FUNCTION Convert_LWORD_TO_TOD : Hresult
VAR_INPUT
	in : LWORD;
	out : REFERENCE TO TOD;
END_VAR
VAR
	converted : TOD;
END_VAR

converted := LWORD_TO_TOD(in);

IF (TOD_TO_LWORD(converted) <> in) THEN
	Convert_LWORD_TO_TOD := INCOMPATIBLE;
	RETURN;
END_IF

out := converted;

END_FUNCTION

(* stored: Version 1.1.0.1, ProductVersion 3.1.4024.12
   POU Convert_LWORD_TO_TOD: Id {14e11d3a-3f43-428f-a00a-499b7135c48f}, SpecialFunc None *)
